// TIA Portal project "TEST_20191209" (V15.1)

(* hardware
DEVICE "S7-1200 station_1"  S7-1200 Station
   slot 0: "Rack_0"  S7-1200 Rack  Rack  V1.0
   slot 1: "PLC_1"  CPU 1214C DC/DC/DC  6ES7 214-1AG40-0XB0  V4.2
*)

// ===== PLC "PLC_1"  CPU 1214C DC/DC/DC =====

VAR_GLOBAL   // PLC tag table "默认变量表"
   "Q1.0_RUN" AT %Q1.0 : Bool;
   "M8192_START" AT %M8191.0 : Bool;
   "M8192_STOP" AT %M8191.1 : Bool;
   "M8197_RUN" AT %M8191.7 : Bool;
   "I1.0_START" AT %I1.0 : Bool;
   "I1.1_STOP" AT %I1.1 : Bool;
   "TEST_FC_LAD_M0.0" AT %M0.0 : Bool;
   "TEST_FC_LAD_M0.1" AT %M0.1 : Bool;
   "TEST_FC_LAD_M0.2" AT %M0.2 : Bool;
   "TEST_FC_SCL_M1.0" AT %M1.0 : Bool;
   "TEST_FC_SCL_M1.1" AT %M1.1 : Bool;
   "INDEX_MD20" AT %MD20 : DInt;
   "OUT_INDEX_MD24" AT %MD24 : DInt;
   "TEST_RUN" AT %M2.0 : Bool;
   "TEST_STEP" AT %MD10 : DInt;
   "TEST_OUT_Q0.0" AT %Q0.0 : Bool;
   "TEST_OUT_Q0.1" AT %Q0.1 : Bool;
   "TEST_OUT_Q0.2" AT %Q0.2 : Bool;
   "TEST_DELAY" AT %MD14 : DInt;
END_VAR

DATA_BLOCK "DB_S7NET"   // DB1
{ S7_Optimized_Access := 'FALSE' }
VERSION : 0.1
   VAR
      Bool1 : Bool := FALSE;
      Bool2 : Bool;
      Dint1 : DInt;
      Dint2 : DInt := 0;
   END_VAR
BEGIN
END_DATA_BLOCK

DATA_BLOCK "DB_ARRAY"   // DB2
{ S7_Optimized_Access := 'TRUE' }
VERSION : 0.1
   VAR
      ARRAY_BOOL : Array[0..99] of Bool;
      ARRAY_DINT : Array[0..99] of DInt;
      INDEX_DB : DInt;
      OUT_INDEX_DB : DInt;
   END_VAR
BEGIN
END_DATA_BLOCK

DATA_BLOCK "DB_Timers"   // DB100
{ S7_Optimized_Access := 'TRUE' }
VERSION : 0.1
   VAR
      TON : Array[0..99] of IEC_TIMER;
   END_VAR
BEGIN
END_DATA_BLOCK

// folder: System blocks/Program resources

DATA_BLOCK "IEC_Timer_0_DB_1"   // DB101
{ S7_Optimized_Access := 'TRUE' }
AUTHOR : Simatic
FAMILY : IEC
NAME : IEC_TMR
VERSION : 1.0
// stored: InstanceOfName IEC_TIMER
"IEC_TIMER"
BEGIN
END_DATA_BLOCK

// folder: (top level)

FUNCTION "TEST_FC_LAD" : Void   // FC1, LAD
{ S7_Optimized_Access := 'TRUE' }
VERSION : 0.1
BEGIN

REGION Network 1
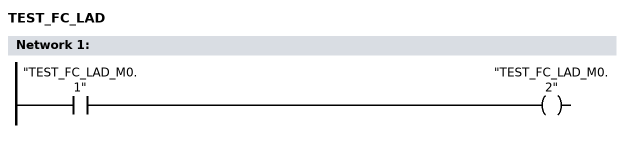
   RUNG wire#powerrail
      Contact( "TEST_FC_LAD_M0.1" )
      Coil( "TEST_FC_LAD_M0.2" )
   END_RUNG
   // the same network as SCL:
   "TEST_FC_LAD_M0.2" := "TEST_FC_LAD_M0.1";
END_REGION
END_FUNCTION

FUNCTION "TEST_FC_SCL" : Void   // FC2, SCL
{ S7_Optimized_Access := 'TRUE' }
VERSION : 0.1
BEGIN
   "TEST_FC_SCL_M1.1" := "TEST_FC_SCL_M1.0";
END_FUNCTION

FUNCTION "TEST_FC_FBD" : Void   // FC3, FBD
{ S7_Optimized_Access := 'TRUE' }
VERSION : 0.1
BEGIN

REGION Network 1
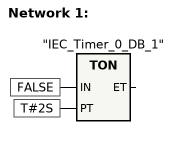
   "IEC_Timer_0_DB_1".TON(IN := FALSE, PT := T#2S);
END_REGION
END_FUNCTION

FUNCTION "TEST_ACTION" : Void   // FC4, LAD
{ S7_Optimized_Access := 'TRUE' }
VERSION : 0.1
   VAR_TEMP   // added for the SCL form of the ladder/FBD networks
      _w1 : Bool;
   END_VAR
BEGIN

REGION Network 1
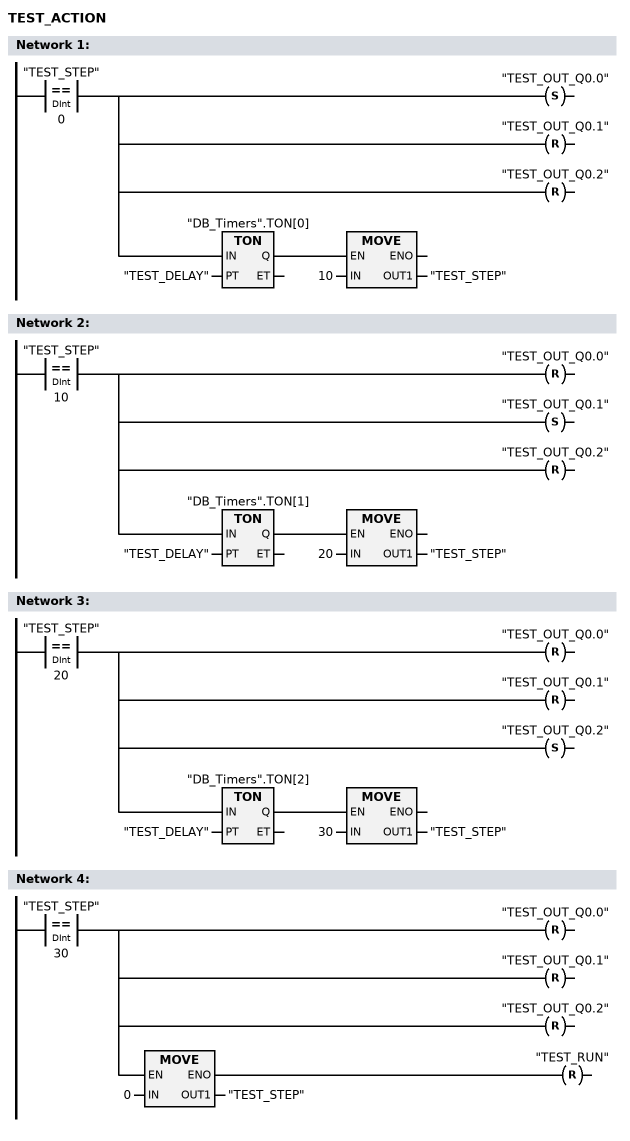
   #_w1 := "TEST_STEP" = 0;
   IF #_w1 THEN
       "TEST_OUT_Q0.0" := TRUE;
       "TEST_OUT_Q0.1" := FALSE;
       "TEST_OUT_Q0.2" := FALSE;
   END_IF;
   "DB_Timers".TON[0].TON(IN := #_w1, PT := "TEST_DELAY");
   IF "DB_Timers".TON[0].Q THEN "TEST_STEP" := 10; END_IF;
END_REGION

REGION Network 2
   #_w1 := "TEST_STEP" = 10;
   IF #_w1 THEN
       "TEST_OUT_Q0.0" := FALSE;
       "TEST_OUT_Q0.1" := TRUE;
       "TEST_OUT_Q0.2" := FALSE;
   END_IF;
   "DB_Timers".TON[1].TON(IN := #_w1, PT := "TEST_DELAY");
   IF "DB_Timers".TON[1].Q THEN "TEST_STEP" := 20; END_IF;
END_REGION

REGION Network 3
   #_w1 := "TEST_STEP" = 20;
   IF #_w1 THEN
       "TEST_OUT_Q0.0" := FALSE;
       "TEST_OUT_Q0.1" := FALSE;
       "TEST_OUT_Q0.2" := TRUE;
   END_IF;
   "DB_Timers".TON[2].TON(IN := #_w1, PT := "TEST_DELAY");
   IF "DB_Timers".TON[2].Q THEN "TEST_STEP" := 30; END_IF;
END_REGION

REGION Network 4
   RUNG wire#powerrail
      { S7_Templates := "SrcType := DInt" } EQ_Contact(in1 := "TEST_STEP", in2 := 30)
      wire#w1
      R_Coil( "TEST_OUT_Q0.0" )
   END_RUNG
   RUNG wire#w1
      R_Coil( "TEST_OUT_Q0.1" )
   END_RUNG
   RUNG wire#w1
      R_Coil( "TEST_OUT_Q0.2" )
   END_RUNG
   RUNG wire#w1
      Move(in := 0, out1 => "TEST_STEP")
      R_Coil( "TEST_RUN" )
   END_RUNG
   // the same network as SCL:
   IF "TEST_STEP" = 30 THEN
       "TEST_OUT_Q0.0" := FALSE;
       "TEST_OUT_Q0.1" := FALSE;
       "TEST_OUT_Q0.2" := FALSE;
   END_IF;
   #_w1 := "TEST_STEP" = 30;
   IF #_w1 THEN
       "TEST_STEP" := 0;
       "TEST_RUN" := FALSE;
   END_IF;
END_REGION
END_FUNCTION

ORGANIZATION_BLOCK "Main"   // OB1, LAD, ProgramCycle
TITLE = "Main Program Sweep (Cycle)"
{ S7_Optimized_Access := 'TRUE' }
VERSION : 0.1
   VAR_INPUT
      Initial_Call : Bool;   // Initial call of this OB
      Remanence : Bool;   // =True, if remanent data are available
   END_VAR
   VAR_TEMP   // added for the SCL form of the ladder/FBD networks
      _w1 : Bool;
   END_VAR
BEGIN

REGION Network 1
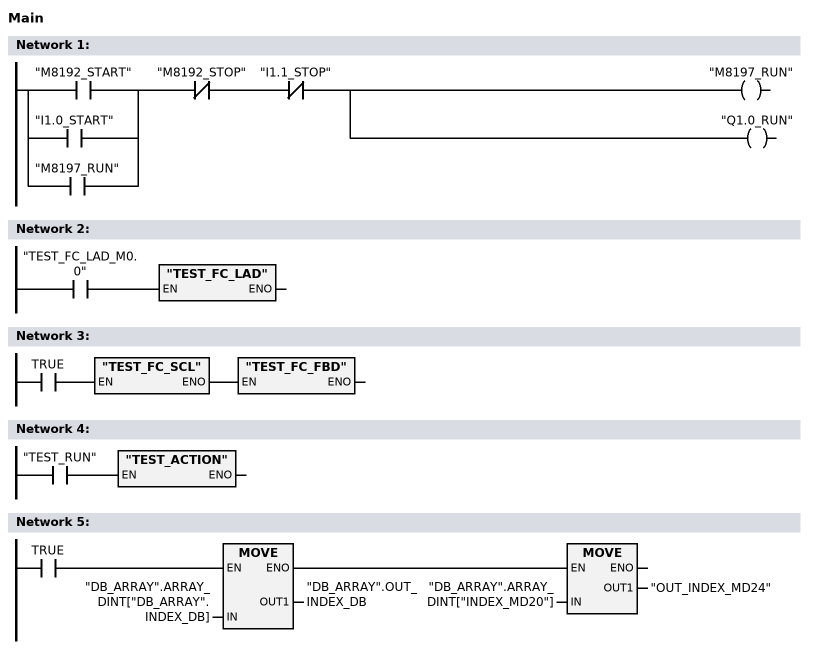
   RUNG wire#powerrail
      Contact( "M8192_START" )
      wire#w1
      I_Contact( "M8192_STOP" )
      I_Contact( "I1.1_STOP" )
      wire#w2
      Coil( "M8197_RUN" )
   END_RUNG
   RUNG wire#powerrail
      Contact( "I1.0_START" )
   END_RUNG wire#w1
   RUNG wire#powerrail
      Contact( "M8197_RUN" )
   END_RUNG wire#w1
   RUNG wire#w2
      Coil( "Q1.0_RUN" )
   END_RUNG
   // the same network as SCL:
   "M8197_RUN" := ("M8192_START" OR "I1.0_START" OR "M8197_RUN") AND NOT "M8192_STOP" AND NOT "I1.1_STOP";
   "Q1.0_RUN" := "M8197_RUN";
END_REGION

REGION Network 2
   RUNG wire#powerrail
      Contact( "TEST_FC_LAD_M0.0" )
      "TEST_FC_LAD"()
   END_RUNG
   // the same network as SCL:
   IF "TEST_FC_LAD_M0.0" THEN "TEST_FC_LAD"(); END_IF;
END_REGION

REGION Network 3
   RUNG wire#powerrail
      Contact( TRUE )
      "TEST_FC_SCL"()
      "TEST_FC_FBD"()
   END_RUNG
   // the same network as SCL:
   "TEST_FC_SCL"(EN := TRUE, ENO => #_w1);
   IF #_w1 THEN "TEST_FC_FBD"(); END_IF;
END_REGION

REGION Network 4
   RUNG wire#powerrail
      Contact( "TEST_RUN" )
      "TEST_ACTION"()
   END_RUNG
   // the same network as SCL:
   IF "TEST_RUN" THEN "TEST_ACTION"(); END_IF;
END_REGION

REGION Network 5
   RUNG wire#powerrail
      Contact( TRUE )
      Move(in := "DB_ARRAY".ARRAY_DINT["DB_ARRAY".INDEX_DB], out1 => "DB_ARRAY".OUT_INDEX_DB)
      Move(in := "DB_ARRAY".ARRAY_DINT["INDEX_MD20"], out1 => "OUT_INDEX_MD24")
   END_RUNG
   // the same network as SCL:
   IF TRUE THEN
       "DB_ARRAY".OUT_INDEX_DB := "DB_ARRAY".ARRAY_DINT["DB_ARRAY".INDEX_DB];
       "OUT_INDEX_MD24" := "DB_ARRAY".ARRAY_DINT["INDEX_MD20"];
   END_IF;
END_REGION
END_ORGANIZATION_BLOCK